// Brief: Mounting Endoscope
FUNCTION_BLOCK PUBLIC FB_SlaveCtrlMountScope EXTENDS FB_SlaveArmCtrlBase
VAR_INPUT
END_VAR
VAR_OUTPUT
END_VAR
VAR
END_VAR

METHOD PUBLIC init : BOOL
VAR_IN_OUT CONSTANT
	i_slaveArm	:FB_SlaveArm;
END_VAR
VAR_IN_OUT 
	r_slaveArmCtrlCmd :ST_SlaveArmCtrlCmds;
END_VAR
// check if to hold the command joint position unchanged
m_holdLastCmds := checkToHoldLastCmds(r_slaveArmCtrlCmd, i_slaveArm);

//init
SUPER^.Init(i_slaveArm,r_slaveArmCtrlCmd);
END_METHOD

END_FUNCTION_BLOCK

(* stored: Version 1.1.0.1, ProductVersion 3.1.4024.11
   POU FB_SlaveCtrlMountScope: Id {6d193be5-4a80-4dd6-a6a8-788f7e960ba3}, SpecialFunc None
   Method init: Id {104a1427-1bba-4e19-a683-ee9a7810b475} *)
